Fanuc KAREL source: VOL_SPACE.kl

PROGRAM T
%NOLOCKGROUP
VAR
 v0 : STRING[40]
 v1 : INTEGER
 v2 : INTEGER
 v3 : STRING[40]
BEGIN
 VOL_SPACE(v0, v1, v2, v3)
END T
